ABB RAPID module: robotcode.MOD

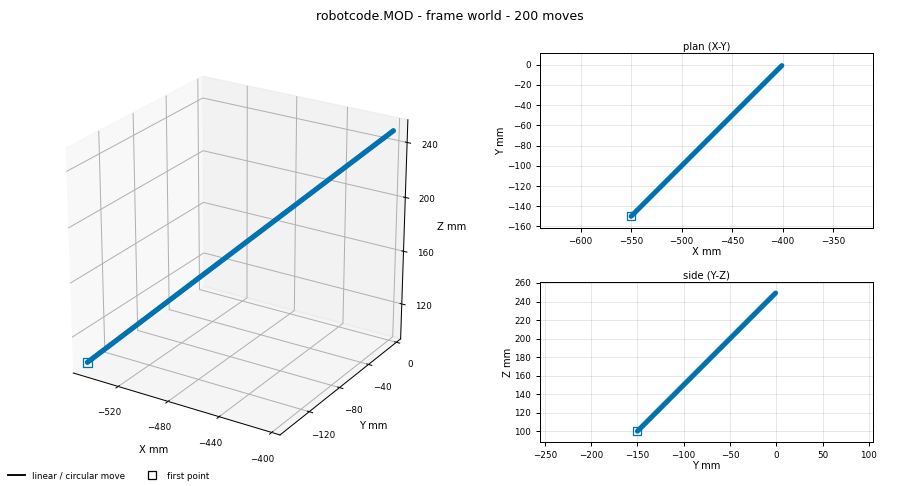
[picture p0: tool path of robotcode.MOD in frame world, 200 of 201 moves have a stored position in this frame; points joined in program order, loops and branches not executed]
MODULE MainModule
PERS tooldata Servo:=[TRUE,[[0,0,114.2],[1,0,0,0]],[0.215,[8.7,12.3,49.2],[1,0,0,0],0.00021,0.00024,0.00009]];
PERS tooldata tObject:=[TRUE,[[0,0,130],[0.707106781,-0.707106781,0,0]],[0.215,[8.7,12.3,49.2],[1,0,0,0],0.00021,0.00024,0.00009]];
PERS wobjdata handpos:= [FALSE,TRUE,"",[[-400,0,250],[1,0,0,0]],[[0,0,0],[1,0,0,0]]];
    PROC main()
        ConfL\Off;
        SingArea\Wrist;
        !Startpos
        MoveAbsJ [[0.441359,-16.418,10.8814,2.79121,60.2034,-14.3875],[168.362,9E+09,9E+09,9E+09,9E+09,9E+09]] \NoEOffs, v1000, fine, wi_tGripper;
        path;
    ENDPROC
    PROC path()

VAR robtarget t0 := [[-150.0, -150.0, -150.0], [0, -1, 0, 0], [0,0,-1,4], [-96,9E+09,9E+09,9E+09,9E+09,9E+09]];
VAR robtarget t1 := [[-149.25, -149.25, -149.25], [0, -1, 0, 0], [0,0,-1,4], [-96,9E+09,9E+09,9E+09,9E+09,9E+09]];
VAR robtarget t2 := [[-148.5, -148.5, -148.5], [0, -1, 0, 0], [0,0,-1,4], [-96,9E+09,9E+09,9E+09,9E+09,9E+09]];
VAR robtarget t3 := [[-147.75, -147.75, -147.75], [0, -1, 0, 0], [0,0,-1,4], [-96,9E+09,9E+09,9E+09,9E+09,9E+09]];
VAR robtarget t4 := [[-147.0, -147.0, -147.0], [0, -1, 0, 0], [0,0,-1,4], [-96,9E+09,9E+09,9E+09,9E+09,9E+09]];
VAR robtarget t5 := [[-146.25, -146.25, -146.25], [0, -1, 0, 0], [0,0,-1,4], [-96,9E+09,9E+09,9E+09,9E+09,9E+09]];
VAR robtarget t6 := [[-145.5, -145.5, -145.5], [0, -1, 0, 0], [0,0,-1,4], [-96,9E+09,9E+09,9E+09,9E+09,9E+09]];
VAR robtarget t7 := [[-144.75, -144.75, -144.75], [0, -1, 0, 0], [0,0,-1,4], [-96,9E+09,9E+09,9E+09,9E+09,9E+09]];
VAR robtarget t8 := [[-144.0, -144.0, -144.0], [0, -1, 0, 0], [0,0,-1,4], [-96,9E+09,9E+09,9E+09,9E+09,9E+09]];
VAR robtarget t9 := [[-143.25, -143.25, -143.25], [0, -1, 0, 0], [0,0,-1,4], [-96,9E+09,9E+09,9E+09,9E+09,9E+09]];
VAR robtarget t10 := [[-142.5, -142.5, -142.5], [0, -1, 0, 0], [0,0,-1,4], [-96,9E+09,9E+09,9E+09,9E+09,9E+09]];
VAR robtarget t11 := [[-141.75, -141.75, -141.75], [0, -1, 0, 0], [0,0,-1,4], [-96,9E+09,9E+09,9E+09,9E+09,9E+09]];
VAR robtarget t12 := [[-141.0, -141.0, -141.0], [0, -1, 0, 0], [0,0,-1,4], [-96,9E+09,9E+09,9E+09,9E+09,9E+09]];
VAR robtarget t13 := [[-140.25, -140.25, -140.25], [0, -1, 0, 0], [0,0,-1,4], [-96,9E+09,9E+09,9E+09,9E+09,9E+09]];
VAR robtarget t14 := [[-139.49999999999997, -139.49999999999997, -139.49999999999997], [0, -1, 0, 0], [0,0,-1,4], [-96,9E+09,9E+09,9E+09,9E+09,9E+09]];
VAR robtarget t15 := [[-138.74999999999997, -138.74999999999997, -138.74999999999997], [0, -1, 0, 0], [0,0,-1,4], [-96,9E+09,9E+09,9E+09,9E+09,9E+09]];
VAR robtarget t16 := [[-137.99999999999997, -137.99999999999997, -137.99999999999997], [0, -1, 0, 0], [0,0,-1,4], [-96,9E+09,9E+09,9E+09,9E+09,9E+09]];
VAR robtarget t17 := [[-137.24999999999997, -137.24999999999997, -137.24999999999997], [0, -1, 0, 0], [0,0,-1,4], [-96,9E+09,9E+09,9E+09,9E+09,9E+09]];
VAR robtarget t18 := [[-136.49999999999997, -136.49999999999997, -136.49999999999997], [0, -1, 0, 0], [0,0,-1,4], [-96,9E+09,9E+09,9E+09,9E+09,9E+09]];
VAR robtarget t19 := [[-135.74999999999997, -135.74999999999997, -135.74999999999997], [0, -1, 0, 0], [0,0,-1,4], [-96,9E+09,9E+09,9E+09,9E+09,9E+09]];
VAR robtarget t20 := [[-135.0, -135.0, -135.0], [0, -1, 0, 0], [0,0,-1,4], [-96,9E+09,9E+09,9E+09,9E+09,9E+09]];
VAR robtarget t21 := [[-134.24999999999997, -134.24999999999997, -134.24999999999997], [0, -1, 0, 0], [0,0,-1,4], [-96,9E+09,9E+09,9E+09,9E+09,9E+09]];
VAR robtarget t22 := [[-133.5, -133.5, -133.5], [0, -1, 0, 0], [0,0,-1,4], [-96,9E+09,9E+09,9E+09,9E+09,9E+09]];
VAR robtarget t23 := [[-132.74999999999997, -132.74999999999997, -132.74999999999997], [0, -1, 0, 0], [0,0,-1,4], [-96,9E+09,9E+09,9E+09,9E+09,9E+09]];
VAR robtarget t24 := [[-132.0, -132.0, -132.0], [0, -1, 0, 0], [0,0,-1,4], [-96,9E+09,9E+09,9E+09,9E+09,9E+09]];
VAR robtarget t25 := [[-131.25, -131.25, -131.25], [0, -1, 0, 0], [0,0,-1,4], [-96,9E+09,9E+09,9E+09,9E+09,9E+09]];
VAR robtarget t26 := [[-130.5, -130.5, -130.5], [0, -1, 0, 0], [0,0,-1,4], [-96,9E+09,9E+09,9E+09,9E+09,9E+09]];
VAR robtarget t27 := [[-129.75, -129.75, -129.75], [0, -1, 0, 0], [0,0,-1,4], [-96,9E+09,9E+09,9E+09,9E+09,9E+09]];
VAR robtarget t28 := [[-129.0, -129.0, -129.0], [0, -1, 0, 0], [0,0,-1,4], [-96,9E+09,9E+09,9E+09,9E+09,9E+09]];
VAR robtarget t29 := [[-128.25, -128.25, -128.25], [0, -1, 0, 0], [0,0,-1,4], [-96,9E+09,9E+09,9E+09,9E+09,9E+09]];
VAR robtarget t30 := [[-127.5, -127.5, -127.5], [0, -1, 0, 0], [0,0,-1,4], [-96,9E+09,9E+09,9E+09,9E+09,9E+09]];
VAR robtarget t31 := [[-126.75, -126.75, -126.75], [0, -1, 0, 0], [0,0,-1,4], [-96,9E+09,9E+09,9E+09,9E+09,9E+09]];
VAR robtarget t32 := [[-126.0, -126.0, -126.0], [0, -1, 0, 0], [0,0,-1,4], [-96,9E+09,9E+09,9E+09,9E+09,9E+09]];
VAR robtarget t33 := [[-125.25, -125.25, -125.25], [0, -1, 0, 0], [0,0,-1,4], [-96,9E+09,9E+09,9E+09,9E+09,9E+09]];
VAR robtarget t34 := [[-124.5, -124.5, -124.5], [0, -1, 0, 0], [0,0,-1,4], [-96,9E+09,9E+09,9E+09,9E+09,9E+09]];
VAR robtarget t35 := [[-123.75, -123.75, -123.75], [0, -1, 0, 0], [0,0,-1,4], [-96,9E+09,9E+09,9E+09,9E+09,9E+09]];
VAR robtarget t36 := [[-123.0, -123.0, -123.0], [0, -1, 0, 0], [0,0,-1,4], [-96,9E+09,9E+09,9E+09,9E+09,9E+09]];
VAR robtarget t37 := [[-122.25, -122.25, -122.25], [0, -1, 0, 0], [0,0,-1,4], [-96,9E+09,9E+09,9E+09,9E+09,9E+09]];
VAR robtarget t38 := [[-121.5, -121.5, -121.5], [0, -1, 0, 0], [0,0,-1,4], [-96,9E+09,9E+09,9E+09,9E+09,9E+09]];
VAR robtarget t39 := [[-120.75, -120.75, -120.75], [0, -1, 0, 0], [0,0,-1,4], [-96,9E+09,9E+09,9E+09,9E+09,9E+09]];
VAR robtarget t40 := [[-120.0, -120.0, -120.0], [0, -1, 0, 0], [0,0,-1,4], [-96,9E+09,9E+09,9E+09,9E+09,9E+09]];
VAR robtarget t41 := [[-119.25, -119.25, -119.25], [0, -1, 0, 0], [0,0,-1,4], [-96,9E+09,9E+09,9E+09,9E+09,9E+09]];
VAR robtarget t42 := [[-118.5, -118.5, -118.5], [0, -1, 0, 0], [0,0,-1,4], [-96,9E+09,9E+09,9E+09,9E+09,9E+09]];
VAR robtarget t43 := [[-117.75, -117.75, -117.75], [0, -1, 0, 0], [0,0,-1,4], [-96,9E+09,9E+09,9E+09,9E+09,9E+09]];
VAR robtarget t44 := [[-117.0, -117.0, -117.0], [0, -1, 0, 0], [0,0,-1,4], [-96,9E+09,9E+09,9E+09,9E+09,9E+09]];
VAR robtarget t45 := [[-116.24999999999999, -116.24999999999999, -116.24999999999999], [0, -1, 0, 0], [0,0,-1,4], [-96,9E+09,9E+09,9E+09,9E+09,9E+09]];
VAR robtarget t46 := [[-115.49999999999999, -115.49999999999999, -115.49999999999999], [0, -1, 0, 0], [0,0,-1,4], [-96,9E+09,9E+09,9E+09,9E+09,9E+09]];
VAR robtarget t47 := [[-114.74999999999999, -114.74999999999999, -114.74999999999999], [0, -1, 0, 0], [0,0,-1,4], [-96,9E+09,9E+09,9E+09,9E+09,9E+09]];
VAR robtarget t48 := [[-113.99999999999999, -113.99999999999999, -113.99999999999999], [0, -1, 0, 0], [0,0,-1,4], [-96,9E+09,9E+09,9E+09,9E+09,9E+09]];
VAR robtarget t49 := [[-113.24999999999999, -113.24999999999999, -113.24999999999999], [0, -1, 0, 0], [0,0,-1,4], [-96,9E+09,9E+09,9E+09,9E+09,9E+09]];
VAR robtarget t50 := [[-112.49999999999999, -112.49999999999999, -112.49999999999999], [0, -1, 0, 0], [0,0,-1,4], [-96,9E+09,9E+09,9E+09,9E+09,9E+09]];
VAR robtarget t51 := [[-111.74999999999999, -111.74999999999999, -111.74999999999999], [0, -1, 0, 0], [0,0,-1,4], [-96,9E+09,9E+09,9E+09,9E+09,9E+09]];
VAR robtarget t52 := [[-110.99999999999999, -110.99999999999999, -110.99999999999999], [0, -1, 0, 0], [0,0,-1,4], [-96,9E+09,9E+09,9E+09,9E+09,9E+09]];
VAR robtarget t53 := [[-110.24999999999999, -110.24999999999999, -110.24999999999999], [0, -1, 0, 0], [0,0,-1,4], [-96,9E+09,9E+09,9E+09,9E+09,9E+09]];
VAR robtarget t54 := [[-109.49999999999999, -109.49999999999999, -109.49999999999999], [0, -1, 0, 0], [0,0,-1,4], [-96,9E+09,9E+09,9E+09,9E+09,9E+09]];
VAR robtarget t55 := [[-108.74999999999999, -108.74999999999999, -108.74999999999999], [0, -1, 0, 0], [0,0,-1,4], [-96,9E+09,9E+09,9E+09,9E+09,9E+09]];
VAR robtarget t56 := [[-107.99999999999999, -107.99999999999999, -107.99999999999999], [0, -1, 0, 0], [0,0,-1,4], [-96,9E+09,9E+09,9E+09,9E+09,9E+09]];
VAR robtarget t57 := [[-107.24999999999999, -107.24999999999999, -107.24999999999999], [0, -1, 0, 0], [0,0,-1,4], [-96,9E+09,9E+09,9E+09,9E+09,9E+09]];
VAR robtarget t58 := [[-106.49999999999999, -106.49999999999999, -106.49999999999999], [0, -1, 0, 0], [0,0,-1,4], [-96,9E+09,9E+09,9E+09,9E+09,9E+09]];
VAR robtarget t59 := [[-105.75000000000001, -105.75000000000001, -105.75000000000001], [0, -1, 0, 0], [0,0,-1,4], [-96,9E+09,9E+09,9E+09,9E+09,9E+09]];
VAR robtarget t60 := [[-104.99999999999999, -104.99999999999999, -104.99999999999999], [0, -1, 0, 0], [0,0,-1,4], [-96,9E+09,9E+09,9E+09,9E+09,9E+09]];
VAR robtarget t61 := [[-104.25000000000001, -104.25000000000001, -104.25000000000001], [0, -1, 0, 0], [0,0,-1,4], [-96,9E+09,9E+09,9E+09,9E+09,9E+09]];
VAR robtarget t62 := [[-103.49999999999999, -103.49999999999999, -103.49999999999999], [0, -1, 0, 0], [0,0,-1,4], [-96,9E+09,9E+09,9E+09,9E+09,9E+09]];
VAR robtarget t63 := [[-102.75000000000001, -102.75000000000001, -102.75000000000001], [0, -1, 0, 0], [0,0,-1,4], [-96,9E+09,9E+09,9E+09,9E+09,9E+09]];
VAR robtarget t64 := [[-101.99999999999999, -101.99999999999999, -101.99999999999999], [0, -1, 0, 0], [0,0,-1,4], [-96,9E+09,9E+09,9E+09,9E+09,9E+09]];
VAR robtarget t65 := [[-101.25, -101.25, -101.25], [0, -1, 0, 0], [0,0,-1,4], [-96,9E+09,9E+09,9E+09,9E+09,9E+09]];
VAR robtarget t66 := [[-100.49999999999997, -100.49999999999997, -100.49999999999997], [0, -1, 0, 0], [0,0,-1,4], [-96,9E+09,9E+09,9E+09,9E+09,9E+09]];
VAR robtarget t67 := [[-99.75, -99.75, -99.75], [0, -1, 0, 0], [0,0,-1,4], [-96,9E+09,9E+09,9E+09,9E+09,9E+09]];
VAR robtarget t68 := [[-98.99999999999997, -98.99999999999997, -98.99999999999997], [0, -1, 0, 0], [0,0,-1,4], [-96,9E+09,9E+09,9E+09,9E+09,9E+09]];
VAR robtarget t69 := [[-98.25, -98.25, -98.25], [0, -1, 0, 0], [0,0,-1,4], [-96,9E+09,9E+09,9E+09,9E+09,9E+09]];
VAR robtarget t70 := [[-97.5, -97.5, -97.5], [0, -1, 0, 0], [0,0,-1,4], [-96,9E+09,9E+09,9E+09,9E+09,9E+09]];
VAR robtarget t71 := [[-96.75, -96.75, -96.75], [0, -1, 0, 0], [0,0,-1,4], [-96,9E+09,9E+09,9E+09,9E+09,9E+09]];
VAR robtarget t72 := [[-96.0, -96.0, -96.0], [0, -1, 0, 0], [0,0,-1,4], [-96,9E+09,9E+09,9E+09,9E+09,9E+09]];
VAR robtarget t73 := [[-95.25, -95.25, -95.25], [0, -1, 0, 0], [0,0,-1,4], [-96,9E+09,9E+09,9E+09,9E+09,9E+09]];
VAR robtarget t74 := [[-94.5, -94.5, -94.5], [0, -1, 0, 0], [0,0,-1,4], [-96,9E+09,9E+09,9E+09,9E+09,9E+09]];
VAR robtarget t75 := [[-93.75, -93.75, -93.75], [0, -1, 0, 0], [0,0,-1,4], [-96,9E+09,9E+09,9E+09,9E+09,9E+09]];
VAR robtarget t76 := [[-93.0, -93.0, -93.0], [0, -1, 0, 0], [0,0,-1,4], [-96,9E+09,9E+09,9E+09,9E+09,9E+09]];
VAR robtarget t77 := [[-92.25, -92.25, -92.25], [0, -1, 0, 0], [0,0,-1,4], [-96,9E+09,9E+09,9E+09,9E+09,9E+09]];
VAR robtarget t78 := [[-91.5, -91.5, -91.5], [0, -1, 0, 0], [0,0,-1,4], [-96,9E+09,9E+09,9E+09,9E+09,9E+09]];
VAR robtarget t79 := [[-90.75, -90.75, -90.75], [0, -1, 0, 0], [0,0,-1,4], [-96,9E+09,9E+09,9E+09,9E+09,9E+09]];
VAR robtarget t80 := [[-90.0, -90.0, -90.0], [0, -1, 0, 0], [0,0,-1,4], [-96,9E+09,9E+09,9E+09,9E+09,9E+09]];
VAR robtarget t81 := [[-89.25, -89.25, -89.25], [0, -1, 0, 0], [0,0,-1,4], [-96,9E+09,9E+09,9E+09,9E+09,9E+09]];
VAR robtarget t82 := [[-88.5, -88.5, -88.5], [0, -1, 0, 0], [0,0,-1,4], [-96,9E+09,9E+09,9E+09,9E+09,9E+09]];
VAR robtarget t83 := [[-87.75, -87.75, -87.75], [0, -1, 0, 0], [0,0,-1,4], [-96,9E+09,9E+09,9E+09,9E+09,9E+09]];
VAR robtarget t84 := [[-87.0, -87.0, -87.0], [0, -1, 0, 0], [0,0,-1,4], [-96,9E+09,9E+09,9E+09,9E+09,9E+09]];
VAR robtarget t85 := [[-86.25, -86.25, -86.25], [0, -1, 0, 0], [0,0,-1,4], [-96,9E+09,9E+09,9E+09,9E+09,9E+09]];
VAR robtarget t86 := [[-85.49999999999999, -85.49999999999999, -85.49999999999999], [0, -1, 0, 0], [0,0,-1,4], [-96,9E+09,9E+09,9E+09,9E+09,9E+09]];
VAR robtarget t87 := [[-84.74999999999999, -84.74999999999999, -84.74999999999999], [0, -1, 0, 0], [0,0,-1,4], [-96,9E+09,9E+09,9E+09,9E+09,9E+09]];
VAR robtarget t88 := [[-83.99999999999999, -83.99999999999999, -83.99999999999999], [0, -1, 0, 0], [0,0,-1,4], [-96,9E+09,9E+09,9E+09,9E+09,9E+09]];
VAR robtarget t89 := [[-83.24999999999999, -83.24999999999999, -83.24999999999999], [0, -1, 0, 0], [0,0,-1,4], [-96,9E+09,9E+09,9E+09,9E+09,9E+09]];
VAR robtarget t90 := [[-82.49999999999999, -82.49999999999999, -82.49999999999999], [0, -1, 0, 0], [0,0,-1,4], [-96,9E+09,9E+09,9E+09,9E+09,9E+09]];
VAR robtarget t91 := [[-81.74999999999999, -81.74999999999999, -81.74999999999999], [0, -1, 0, 0], [0,0,-1,4], [-96,9E+09,9E+09,9E+09,9E+09,9E+09]];
VAR robtarget t92 := [[-80.99999999999999, -80.99999999999999, -80.99999999999999], [0, -1, 0, 0], [0,0,-1,4], [-96,9E+09,9E+09,9E+09,9E+09,9E+09]];
VAR robtarget t93 := [[-80.24999999999999, -80.24999999999999, -80.24999999999999], [0, -1, 0, 0], [0,0,-1,4], [-96,9E+09,9E+09,9E+09,9E+09,9E+09]];
VAR robtarget t94 := [[-79.49999999999999, -79.49999999999999, -79.49999999999999], [0, -1, 0, 0], [0,0,-1,4], [-96,9E+09,9E+09,9E+09,9E+09,9E+09]];
VAR robtarget t95 := [[-78.74999999999999, -78.74999999999999, -78.74999999999999], [0, -1, 0, 0], [0,0,-1,4], [-96,9E+09,9E+09,9E+09,9E+09,9E+09]];
VAR robtarget t96 := [[-77.99999999999999, -77.99999999999999, -77.99999999999999], [0, -1, 0, 0], [0,0,-1,4], [-96,9E+09,9E+09,9E+09,9E+09,9E+09]];
VAR robtarget t97 := [[-77.24999999999999, -77.24999999999999, -77.24999999999999], [0, -1, 0, 0], [0,0,-1,4], [-96,9E+09,9E+09,9E+09,9E+09,9E+09]];
VAR robtarget t98 := [[-76.50000000000001, -76.50000000000001, -76.50000000000001], [0, -1, 0, 0], [0,0,-1,4], [-96,9E+09,9E+09,9E+09,9E+09,9E+09]];
VAR robtarget t99 := [[-75.74999999999999, -75.74999999999999, -75.74999999999999], [0, -1, 0, 0], [0,0,-1,4], [-96,9E+09,9E+09,9E+09,9E+09,9E+09]];
VAR robtarget t100 := [[-75.00000000000001, -75.00000000000001, -75.00000000000001], [0, -1, 0, 0], [0,0,-1,4], [-96,9E+09,9E+09,9E+09,9E+09,9E+09]];
VAR robtarget t101 := [[-74.24999999999999, -74.24999999999999, -74.24999999999999], [0, -1, 0, 0], [0,0,-1,4], [-96,9E+09,9E+09,9E+09,9E+09,9E+09]];
VAR robtarget t102 := [[-73.50000000000001, -73.50000000000001, -73.50000000000001], [0, -1, 0, 0], [0,0,-1,4], [-96,9E+09,9E+09,9E+09,9E+09,9E+09]];
VAR robtarget t103 := [[-72.74999999999999, -72.74999999999999, -72.74999999999999], [0, -1, 0, 0], [0,0,-1,4], [-96,9E+09,9E+09,9E+09,9E+09,9E+09]];
VAR robtarget t104 := [[-72.00000000000001, -72.00000000000001, -72.00000000000001], [0, -1, 0, 0], [0,0,-1,4], [-96,9E+09,9E+09,9E+09,9E+09,9E+09]];
VAR robtarget t105 := [[-71.24999999999999, -71.24999999999999, -71.24999999999999], [0, -1, 0, 0], [0,0,-1,4], [-96,9E+09,9E+09,9E+09,9E+09,9E+09]];
VAR robtarget t106 := [[-70.5, -70.5, -70.5], [0, -1, 0, 0], [0,0,-1,4], [-96,9E+09,9E+09,9E+09,9E+09,9E+09]];
VAR robtarget t107 := [[-69.74999999999997, -69.74999999999997, -69.74999999999997], [0, -1, 0, 0], [0,0,-1,4], [-96,9E+09,9E+09,9E+09,9E+09,9E+09]];
VAR robtarget t108 := [[-69.0, -69.0, -69.0], [0, -1, 0, 0], [0,0,-1,4], [-96,9E+09,9E+09,9E+09,9E+09,9E+09]];
VAR robtarget t109 := [[-68.24999999999997, -68.24999999999997, -68.24999999999997], [0, -1, 0, 0], [0,0,-1,4], [-96,9E+09,9E+09,9E+09,9E+09,9E+09]];
VAR robtarget t110 := [[-67.5, -67.5, -67.5], [0, -1, 0, 0], [0,0,-1,4], [-96,9E+09,9E+09,9E+09,9E+09,9E+09]];
VAR robtarget t111 := [[-66.74999999999997, -66.74999999999997, -66.74999999999997], [0, -1, 0, 0], [0,0,-1,4], [-96,9E+09,9E+09,9E+09,9E+09,9E+09]];
VAR robtarget t112 := [[-66.0, -66.0, -66.0], [0, -1, 0, 0], [0,0,-1,4], [-96,9E+09,9E+09,9E+09,9E+09,9E+09]];
VAR robtarget t113 := [[-65.24999999999997, -65.24999999999997, -65.24999999999997], [0, -1, 0, 0], [0,0,-1,4], [-96,9E+09,9E+09,9E+09,9E+09,9E+09]];
VAR robtarget t114 := [[-64.5, -64.5, -64.5], [0, -1, 0, 0], [0,0,-1,4], [-96,9E+09,9E+09,9E+09,9E+09,9E+09]];
VAR robtarget t115 := [[-63.74999999999997, -63.74999999999997, -63.74999999999997], [0, -1, 0, 0], [0,0,-1,4], [-96,9E+09,9E+09,9E+09,9E+09,9E+09]];
VAR robtarget t116 := [[-63.0, -63.0, -63.0], [0, -1, 0, 0], [0,0,-1,4], [-96,9E+09,9E+09,9E+09,9E+09,9E+09]];
VAR robtarget t117 := [[-62.24999999999997, -62.24999999999997, -62.24999999999997], [0, -1, 0, 0], [0,0,-1,4], [-96,9E+09,9E+09,9E+09,9E+09,9E+09]];
VAR robtarget t118 := [[-61.5, -61.5, -61.5], [0, -1, 0, 0], [0,0,-1,4], [-96,9E+09,9E+09,9E+09,9E+09,9E+09]];
VAR robtarget t119 := [[-60.75, -60.75, -60.75], [0, -1, 0, 0], [0,0,-1,4], [-96,9E+09,9E+09,9E+09,9E+09,9E+09]];
VAR robtarget t120 := [[-60.0, -60.0, -60.0], [0, -1, 0, 0], [0,0,-1,4], [-96,9E+09,9E+09,9E+09,9E+09,9E+09]];
VAR robtarget t121 := [[-59.25, -59.25, -59.25], [0, -1, 0, 0], [0,0,-1,4], [-96,9E+09,9E+09,9E+09,9E+09,9E+09]];
VAR robtarget t122 := [[-58.5, -58.5, -58.5], [0, -1, 0, 0], [0,0,-1,4], [-96,9E+09,9E+09,9E+09,9E+09,9E+09]];
VAR robtarget t123 := [[-57.74999999999999, -57.74999999999999, -57.74999999999999], [0, -1, 0, 0], [0,0,-1,4], [-96,9E+09,9E+09,9E+09,9E+09,9E+09]];
VAR robtarget t124 := [[-56.99999999999999, -56.99999999999999, -56.99999999999999], [0, -1, 0, 0], [0,0,-1,4], [-96,9E+09,9E+09,9E+09,9E+09,9E+09]];
VAR robtarget t125 := [[-56.24999999999999, -56.24999999999999, -56.24999999999999], [0, -1, 0, 0], [0,0,-1,4], [-96,9E+09,9E+09,9E+09,9E+09,9E+09]];
VAR robtarget t126 := [[-55.49999999999999, -55.49999999999999, -55.49999999999999], [0, -1, 0, 0], [0,0,-1,4], [-96,9E+09,9E+09,9E+09,9E+09,9E+09]];
VAR robtarget t127 := [[-54.74999999999999, -54.74999999999999, -54.74999999999999], [0, -1, 0, 0], [0,0,-1,4], [-96,9E+09,9E+09,9E+09,9E+09,9E+09]];
VAR robtarget t128 := [[-53.99999999999999, -53.99999999999999, -53.99999999999999], [0, -1, 0, 0], [0,0,-1,4], [-96,9E+09,9E+09,9E+09,9E+09,9E+09]];
VAR robtarget t129 := [[-53.24999999999999, -53.24999999999999, -53.24999999999999], [0, -1, 0, 0], [0,0,-1,4], [-96,9E+09,9E+09,9E+09,9E+09,9E+09]];
VAR robtarget t130 := [[-52.49999999999999, -52.49999999999999, -52.49999999999999], [0, -1, 0, 0], [0,0,-1,4], [-96,9E+09,9E+09,9E+09,9E+09,9E+09]];
VAR robtarget t131 := [[-51.74999999999999, -51.74999999999999, -51.74999999999999], [0, -1, 0, 0], [0,0,-1,4], [-96,9E+09,9E+09,9E+09,9E+09,9E+09]];
VAR robtarget t132 := [[-50.99999999999999, -50.99999999999999, -50.99999999999999], [0, -1, 0, 0], [0,0,-1,4], [-96,9E+09,9E+09,9E+09,9E+09,9E+09]];
VAR robtarget t133 := [[-50.249999999999986, -50.249999999999986, -50.249999999999986], [0, -1, 0, 0], [0,0,-1,4], [-96,9E+09,9E+09,9E+09,9E+09,9E+09]];
VAR robtarget t134 := [[-49.499999999999986, -49.499999999999986, -49.499999999999986], [0, -1, 0, 0], [0,0,-1,4], [-96,9E+09,9E+09,9E+09,9E+09,9E+09]];
VAR robtarget t135 := [[-48.750000000000014, -48.750000000000014, -48.750000000000014], [0, -1, 0, 0], [0,0,-1,4], [-96,9E+09,9E+09,9E+09,9E+09,9E+09]];
VAR robtarget t136 := [[-47.999999999999986, -47.999999999999986, -47.999999999999986], [0, -1, 0, 0], [0,0,-1,4], [-96,9E+09,9E+09,9E+09,9E+09,9E+09]];
VAR robtarget t137 := [[-47.24999999999996, -47.24999999999996, -47.24999999999996], [0, -1, 0, 0], [0,0,-1,4], [-96,9E+09,9E+09,9E+09,9E+09,9E+09]];
VAR robtarget t138 := [[-46.499999999999986, -46.499999999999986, -46.499999999999986], [0, -1, 0, 0], [0,0,-1,4], [-96,9E+09,9E+09,9E+09,9E+09,9E+09]];
VAR robtarget t139 := [[-45.750000000000014, -45.750000000000014, -45.750000000000014], [0, -1, 0, 0], [0,0,-1,4], [-96,9E+09,9E+09,9E+09,9E+09,9E+09]];
VAR robtarget t140 := [[-44.999999999999986, -44.999999999999986, -44.999999999999986], [0, -1, 0, 0], [0,0,-1,4], [-96,9E+09,9E+09,9E+09,9E+09,9E+09]];
VAR robtarget t141 := [[-44.250000000000014, -44.250000000000014, -44.250000000000014], [0, -1, 0, 0], [0,0,-1,4], [-96,9E+09,9E+09,9E+09,9E+09,9E+09]];
VAR robtarget t142 := [[-43.499999999999986, -43.499999999999986, -43.499999999999986], [0, -1, 0, 0], [0,0,-1,4], [-96,9E+09,9E+09,9E+09,9E+09,9E+09]];
VAR robtarget t143 := [[-42.75000000000001, -42.75000000000001, -42.75000000000001], [0, -1, 0, 0], [0,0,-1,4], [-96,9E+09,9E+09,9E+09,9E+09,9E+09]];
VAR robtarget t144 := [[-41.99999999999998, -41.99999999999998, -41.99999999999998], [0, -1, 0, 0], [0,0,-1,4], [-96,9E+09,9E+09,9E+09,9E+09,9E+09]];
VAR robtarget t145 := [[-41.25000000000001, -41.25000000000001, -41.25000000000001], [0, -1, 0, 0], [0,0,-1,4], [-96,9E+09,9E+09,9E+09,9E+09,9E+09]];
VAR robtarget t146 := [[-40.49999999999998, -40.49999999999998, -40.49999999999998], [0, -1, 0, 0], [0,0,-1,4], [-96,9E+09,9E+09,9E+09,9E+09,9E+09]];
VAR robtarget t147 := [[-39.75000000000001, -39.75000000000001, -39.75000000000001], [0, -1, 0, 0], [0,0,-1,4], [-96,9E+09,9E+09,9E+09,9E+09,9E+09]];
VAR robtarget t148 := [[-38.99999999999998, -38.99999999999998, -38.99999999999998], [0, -1, 0, 0], [0,0,-1,4], [-96,9E+09,9E+09,9E+09,9E+09,9E+09]];
VAR robtarget t149 := [[-38.25000000000001, -38.25000000000001, -38.25000000000001], [0, -1, 0, 0], [0,0,-1,4], [-96,9E+09,9E+09,9E+09,9E+09,9E+09]];
VAR robtarget t150 := [[-37.49999999999998, -37.49999999999998, -37.49999999999998], [0, -1, 0, 0], [0,0,-1,4], [-96,9E+09,9E+09,9E+09,9E+09,9E+09]];
VAR robtarget t151 := [[-36.75000000000001, -36.75000000000001, -36.75000000000001], [0, -1, 0, 0], [0,0,-1,4], [-96,9E+09,9E+09,9E+09,9E+09,9E+09]];
VAR robtarget t152 := [[-35.99999999999998, -35.99999999999998, -35.99999999999998], [0, -1, 0, 0], [0,0,-1,4], [-96,9E+09,9E+09,9E+09,9E+09,9E+09]];
VAR robtarget t153 := [[-35.25, -35.25, -35.25], [0, -1, 0, 0], [0,0,-1,4], [-96,9E+09,9E+09,9E+09,9E+09,9E+09]];
VAR robtarget t154 := [[-34.49999999999997, -34.49999999999997, -34.49999999999997], [0, -1, 0, 0], [0,0,-1,4], [-96,9E+09,9E+09,9E+09,9E+09,9E+09]];
VAR robtarget t155 := [[-33.75, -33.75, -33.75], [0, -1, 0, 0], [0,0,-1,4], [-96,9E+09,9E+09,9E+09,9E+09,9E+09]];
VAR robtarget t156 := [[-32.99999999999997, -32.99999999999997, -32.99999999999997], [0, -1, 0, 0], [0,0,-1,4], [-96,9E+09,9E+09,9E+09,9E+09,9E+09]];
VAR robtarget t157 := [[-32.25, -32.25, -32.25], [0, -1, 0, 0], [0,0,-1,4], [-96,9E+09,9E+09,9E+09,9E+09,9E+09]];
VAR robtarget t158 := [[-31.49999999999997, -31.49999999999997, -31.49999999999997], [0, -1, 0, 0], [0,0,-1,4], [-96,9E+09,9E+09,9E+09,9E+09,9E+09]];
VAR robtarget t159 := [[-30.75, -30.75, -30.75], [0, -1, 0, 0], [0,0,-1,4], [-96,9E+09,9E+09,9E+09,9E+09,9E+09]];
VAR robtarget t160 := [[-29.99999999999997, -29.99999999999997, -29.99999999999997], [0, -1, 0, 0], [0,0,-1,4], [-96,9E+09,9E+09,9E+09,9E+09,9E+09]];
VAR robtarget t161 := [[-29.25, -29.25, -29.25], [0, -1, 0, 0], [0,0,-1,4], [-96,9E+09,9E+09,9E+09,9E+09,9E+09]];
VAR robtarget t162 := [[-28.500000000000025, -28.500000000000025, -28.500000000000025], [0, -1, 0, 0], [0,0,-1,4], [-96,9E+09,9E+09,9E+09,9E+09,9E+09]];
VAR robtarget t163 := [[-27.749999999999996, -27.749999999999996, -27.749999999999996], [0, -1, 0, 0], [0,0,-1,4], [-96,9E+09,9E+09,9E+09,9E+09,9E+09]];
VAR robtarget t164 := [[-26.999999999999968, -26.999999999999968, -26.999999999999968], [0, -1, 0, 0], [0,0,-1,4], [-96,9E+09,9E+09,9E+09,9E+09,9E+09]];
VAR robtarget t165 := [[-26.249999999999996, -26.249999999999996, -26.249999999999996], [0, -1, 0, 0], [0,0,-1,4], [-96,9E+09,9E+09,9E+09,9E+09,9E+09]];
VAR robtarget t166 := [[-25.50000000000002, -25.50000000000002, -25.50000000000002], [0, -1, 0, 0], [0,0,-1,4], [-96,9E+09,9E+09,9E+09,9E+09,9E+09]];
VAR robtarget t167 := [[-24.749999999999993, -24.749999999999993, -24.749999999999993], [0, -1, 0, 0], [0,0,-1,4], [-96,9E+09,9E+09,9E+09,9E+09,9E+09]];
VAR robtarget t168 := [[-23.999999999999964, -23.999999999999964, -23.999999999999964], [0, -1, 0, 0], [0,0,-1,4], [-96,9E+09,9E+09,9E+09,9E+09,9E+09]];
VAR robtarget t169 := [[-23.249999999999993, -23.249999999999993, -23.249999999999993], [0, -1, 0, 0], [0,0,-1,4], [-96,9E+09,9E+09,9E+09,9E+09,9E+09]];
VAR robtarget t170 := [[-22.50000000000002, -22.50000000000002, -22.50000000000002], [0, -1, 0, 0], [0,0,-1,4], [-96,9E+09,9E+09,9E+09,9E+09,9E+09]];
VAR robtarget t171 := [[-21.749999999999993, -21.749999999999993, -21.749999999999993], [0, -1, 0, 0], [0,0,-1,4], [-96,9E+09,9E+09,9E+09,9E+09,9E+09]];
VAR robtarget t172 := [[-20.999999999999964, -20.999999999999964, -20.999999999999964], [0, -1, 0, 0], [0,0,-1,4], [-96,9E+09,9E+09,9E+09,9E+09,9E+09]];
VAR robtarget t173 := [[-20.24999999999999, -20.24999999999999, -20.24999999999999], [0, -1, 0, 0], [0,0,-1,4], [-96,9E+09,9E+09,9E+09,9E+09,9E+09]];
VAR robtarget t174 := [[-19.500000000000018, -19.500000000000018, -19.500000000000018], [0, -1, 0, 0], [0,0,-1,4], [-96,9E+09,9E+09,9E+09,9E+09,9E+09]];
VAR robtarget t175 := [[-18.74999999999999, -18.74999999999999, -18.74999999999999], [0, -1, 0, 0], [0,0,-1,4], [-96,9E+09,9E+09,9E+09,9E+09,9E+09]];
VAR robtarget t176 := [[-17.99999999999996, -17.99999999999996, -17.99999999999996], [0, -1, 0, 0], [0,0,-1,4], [-96,9E+09,9E+09,9E+09,9E+09,9E+09]];
VAR robtarget t177 := [[-17.249999999999986, -17.249999999999986, -17.249999999999986], [0, -1, 0, 0], [0,0,-1,4], [-96,9E+09,9E+09,9E+09,9E+09,9E+09]];
VAR robtarget t178 := [[-16.500000000000014, -16.500000000000014, -16.500000000000014], [0, -1, 0, 0], [0,0,-1,4], [-96,9E+09,9E+09,9E+09,9E+09,9E+09]];
VAR robtarget t179 := [[-15.749999999999986, -15.749999999999986, -15.749999999999986], [0, -1, 0, 0], [0,0,-1,4], [-96,9E+09,9E+09,9E+09,9E+09,9E+09]];
VAR robtarget t180 := [[-14.999999999999957, -14.999999999999957, -14.999999999999957], [0, -1, 0, 0], [0,0,-1,4], [-96,9E+09,9E+09,9E+09,9E+09,9E+09]];
VAR robtarget t181 := [[-14.249999999999986, -14.249999999999986, -14.249999999999986], [0, -1, 0, 0], [0,0,-1,4], [-96,9E+09,9E+09,9E+09,9E+09,9E+09]];
VAR robtarget t182 := [[-13.500000000000012, -13.500000000000012, -13.500000000000012], [0, -1, 0, 0], [0,0,-1,4], [-96,9E+09,9E+09,9E+09,9E+09,9E+09]];
VAR robtarget t183 := [[-12.749999999999984, -12.749999999999984, -12.749999999999984], [0, -1, 0, 0], [0,0,-1,4], [-96,9E+09,9E+09,9E+09,9E+09,9E+09]];
VAR robtarget t184 := [[-11.999999999999956, -11.999999999999956, -11.999999999999956], [0, -1, 0, 0], [0,0,-1,4], [-96,9E+09,9E+09,9E+09,9E+09,9E+09]];
VAR robtarget t185 := [[-11.249999999999982, -11.249999999999982, -11.249999999999982], [0, -1, 0, 0], [0,0,-1,4], [-96,9E+09,9E+09,9E+09,9E+09,9E+09]];
VAR robtarget t186 := [[-10.500000000000009, -10.500000000000009, -10.500000000000009], [0, -1, 0, 0], [0,0,-1,4], [-96,9E+09,9E+09,9E+09,9E+09,9E+09]];
VAR robtarget t187 := [[-9.74999999999998, -9.74999999999998, -9.74999999999998], [0, -1, 0, 0], [0,0,-1,4], [-96,9E+09,9E+09,9E+09,9E+09,9E+09]];
VAR robtarget t188 := [[-8.999999999999952, -8.999999999999952, -8.999999999999952], [0, -1, 0, 0], [0,0,-1,4], [-96,9E+09,9E+09,9E+09,9E+09,9E+09]];
VAR robtarget t189 := [[-8.249999999999979, -8.249999999999979, -8.249999999999979], [0, -1, 0, 0], [0,0,-1,4], [-96,9E+09,9E+09,9E+09,9E+09,9E+09]];
VAR robtarget t190 := [[-7.500000000000007, -7.500000000000007, -7.500000000000007], [0, -1, 0, 0], [0,0,-1,4], [-96,9E+09,9E+09,9E+09,9E+09,9E+09]];
VAR robtarget t191 := [[-6.749999999999979, -6.749999999999979, -6.749999999999979], [0, -1, 0, 0], [0,0,-1,4], [-96,9E+09,9E+09,9E+09,9E+09,9E+09]];
VAR robtarget t192 := [[-5.99999999999995, -5.99999999999995, -5.99999999999995], [0, -1, 0, 0], [0,0,-1,4], [-96,9E+09,9E+09,9E+09,9E+09,9E+09]];
VAR robtarget t193 := [[-5.250000000000032, -5.250000000000032, -5.250000000000032], [0, -1, 0, 0], [0,0,-1,4], [-96,9E+09,9E+09,9E+09,9E+09,9E+09]];
VAR robtarget t194 := [[-4.5000000000000036, -4.5000000000000036, -4.5000000000000036], [0, -1, 0, 0], [0,0,-1,4], [-96,9E+09,9E+09,9E+09,9E+09,9E+09]];
VAR robtarget t195 := [[-3.7499999999999756, -3.7499999999999756, -3.7499999999999756], [0, -1, 0, 0], [0,0,-1,4], [-96,9E+09,9E+09,9E+09,9E+09,9E+09]];
VAR robtarget t196 := [[-3.0000000000000027, -3.0000000000000027, -3.0000000000000027], [0, -1, 0, 0], [0,0,-1,4], [-96,9E+09,9E+09,9E+09,9E+09,9E+09]];
VAR robtarget t197 := [[-2.2500000000000298, -2.2500000000000298, -2.2500000000000298], [0, -1, 0, 0], [0,0,-1,4], [-96,9E+09,9E+09,9E+09,9E+09,9E+09]];
VAR robtarget t198 := [[-1.5000000000000013, -1.5000000000000013, -1.5000000000000013], [0, -1, 0, 0], [0,0,-1,4], [-96,9E+09,9E+09,9E+09,9E+09,9E+09]];
VAR robtarget t199 := [[-0.7499999999999729, -0.7499999999999729, -0.7499999999999729], [0, -1, 0, 0], [0,0,-1,4], [-96,9E+09,9E+09,9E+09,9E+09,9E+09]];MoveL t0, v100\V:=100.000, z1, wi_tGripper, \WObj:=handpos;
MoveL t1, v100\V:=100.000, z1, wi_tGripper, \WObj:=handpos;
MoveL t2, v100\V:=100.000, z1, wi_tGripper, \WObj:=handpos;
MoveL t3, v100\V:=100.000, z1, wi_tGripper, \WObj:=handpos;
MoveL t4, v100\V:=100.000, z1, wi_tGripper, \WObj:=handpos;
MoveL t5, v100\V:=100.000, z1, wi_tGripper, \WObj:=handpos;
MoveL t6, v100\V:=100.000, z1, wi_tGripper, \WObj:=handpos;
MoveL t7, v100\V:=100.000, z1, wi_tGripper, \WObj:=handpos;
MoveL t8, v100\V:=100.000, z1, wi_tGripper, \WObj:=handpos;
MoveL t9, v100\V:=100.000, z1, wi_tGripper, \WObj:=handpos;
MoveL t10, v100\V:=100.000, z1, wi_tGripper, \WObj:=handpos;
MoveL t11, v100\V:=100.000, z1, wi_tGripper, \WObj:=handpos;
MoveL t12, v100\V:=100.000, z1, wi_tGripper, \WObj:=handpos;
MoveL t13, v100\V:=100.000, z1, wi_tGripper, \WObj:=handpos;
MoveL t14, v100\V:=100.000, z1, wi_tGripper, \WObj:=handpos;
MoveL t15, v100\V:=100.000, z1, wi_tGripper, \WObj:=handpos;
MoveL t16, v100\V:=100.000, z1, wi_tGripper, \WObj:=handpos;
MoveL t17, v100\V:=100.000, z1, wi_tGripper, \WObj:=handpos;
MoveL t18, v100\V:=100.000, z1, wi_tGripper, \WObj:=handpos;
MoveL t19, v100\V:=100.000, z1, wi_tGripper, \WObj:=handpos;
MoveL t20, v100\V:=100.000, z1, wi_tGripper, \WObj:=handpos;
MoveL t21, v100\V:=100.000, z1, wi_tGripper, \WObj:=handpos;
MoveL t22, v100\V:=100.000, z1, wi_tGripper, \WObj:=handpos;
MoveL t23, v100\V:=100.000, z1, wi_tGripper, \WObj:=handpos;
MoveL t24, v100\V:=100.000, z1, wi_tGripper, \WObj:=handpos;
MoveL t25, v100\V:=100.000, z1, wi_tGripper, \WObj:=handpos;
MoveL t26, v100\V:=100.000, z1, wi_tGripper, \WObj:=handpos;
MoveL t27, v100\V:=100.000, z1, wi_tGripper, \WObj:=handpos;
MoveL t28, v100\V:=100.000, z1, wi_tGripper, \WObj:=handpos;
MoveL t29, v100\V:=100.000, z1, wi_tGripper, \WObj:=handpos;
MoveL t30, v100\V:=100.000, z1, wi_tGripper, \WObj:=handpos;
MoveL t31, v100\V:=100.000, z1, wi_tGripper, \WObj:=handpos;
MoveL t32, v100\V:=100.000, z1, wi_tGripper, \WObj:=handpos;
MoveL t33, v100\V:=100.000, z1, wi_tGripper, \WObj:=handpos;
MoveL t34, v100\V:=100.000, z1, wi_tGripper, \WObj:=handpos;
MoveL t35, v100\V:=100.000, z1, wi_tGripper, \WObj:=handpos;
MoveL t36, v100\V:=100.000, z1, wi_tGripper, \WObj:=handpos;
MoveL t37, v100\V:=100.000, z1, wi_tGripper, \WObj:=handpos;
MoveL t38, v100\V:=100.000, z1, wi_tGripper, \WObj:=handpos;
MoveL t39, v100\V:=100.000, z1, wi_tGripper, \WObj:=handpos;
MoveL t40, v100\V:=100.000, z1, wi_tGripper, \WObj:=handpos;
MoveL t41, v100\V:=100.000, z1, wi_tGripper, \WObj:=handpos;
MoveL t42, v100\V:=100.000, z1, wi_tGripper, \WObj:=handpos;
MoveL t43, v100\V:=100.000, z1, wi_tGripper, \WObj:=handpos;
MoveL t44, v100\V:=100.000, z1, wi_tGripper, \WObj:=handpos;
MoveL t45, v100\V:=100.000, z1, wi_tGripper, \WObj:=handpos;
MoveL t46, v100\V:=100.000, z1, wi_tGripper, \WObj:=handpos;
MoveL t47, v100\V:=100.000, z1, wi_tGripper, \WObj:=handpos;
MoveL t48, v100\V:=100.000, z1, wi_tGripper, \WObj:=handpos;
MoveL t49, v100\V:=100.000, z1, wi_tGripper, \WObj:=handpos;
MoveL t50, v100\V:=100.000, z1, wi_tGripper, \WObj:=handpos;
MoveL t51, v100\V:=100.000, z1, wi_tGripper, \WObj:=handpos;
MoveL t52, v100\V:=100.000, z1, wi_tGripper, \WObj:=handpos;
MoveL t53, v100\V:=100.000, z1, wi_tGripper, \WObj:=handpos;
MoveL t54, v100\V:=100.000, z1, wi_tGripper, \WObj:=handpos;
MoveL t55, v100\V:=100.000, z1, wi_tGripper, \WObj:=handpos;
MoveL t56, v100\V:=100.000, z1, wi_tGripper, \WObj:=handpos;
MoveL t57, v100\V:=100.000, z1, wi_tGripper, \WObj:=handpos;
MoveL t58, v100\V:=100.000, z1, wi_tGripper, \WObj:=handpos;
MoveL t59, v100\V:=100.000, z1, wi_tGripper, \WObj:=handpos;
MoveL t60, v100\V:=100.000, z1, wi_tGripper, \WObj:=handpos;
MoveL t61, v100\V:=100.000, z1, wi_tGripper, \WObj:=handpos;
MoveL t62, v100\V:=100.000, z1, wi_tGripper, \WObj:=handpos;
MoveL t63, v100\V:=100.000, z1, wi_tGripper, \WObj:=handpos;
MoveL t64, v100\V:=100.000, z1, wi_tGripper, \WObj:=handpos;
MoveL t65, v100\V:=100.000, z1, wi_tGripper, \WObj:=handpos;
MoveL t66, v100\V:=100.000, z1, wi_tGripper, \WObj:=handpos;
MoveL t67, v100\V:=100.000, z1, wi_tGripper, \WObj:=handpos;
MoveL t68, v100\V:=100.000, z1, wi_tGripper, \WObj:=handpos;
MoveL t69, v100\V:=100.000, z1, wi_tGripper, \WObj:=handpos;
MoveL t70, v100\V:=100.000, z1, wi_tGripper, \WObj:=handpos;
MoveL t71, v100\V:=100.000, z1, wi_tGripper, \WObj:=handpos;
MoveL t72, v100\V:=100.000, z1, wi_tGripper, \WObj:=handpos;
MoveL t73, v100\V:=100.000, z1, wi_tGripper, \WObj:=handpos;
MoveL t74, v100\V:=100.000, z1, wi_tGripper, \WObj:=handpos;
MoveL t75, v100\V:=100.000, z1, wi_tGripper, \WObj:=handpos;
MoveL t76, v100\V:=100.000, z1, wi_tGripper, \WObj:=handpos;
MoveL t77, v100\V:=100.000, z1, wi_tGripper, \WObj:=handpos;
MoveL t78, v100\V:=100.000, z1, wi_tGripper, \WObj:=handpos;
MoveL t79, v100\V:=100.000, z1, wi_tGripper, \WObj:=handpos;
MoveL t80, v100\V:=100.000, z1, wi_tGripper, \WObj:=handpos;
MoveL t81, v100\V:=100.000, z1, wi_tGripper, \WObj:=handpos;
MoveL t82, v100\V:=100.000, z1, wi_tGripper, \WObj:=handpos;
MoveL t83, v100\V:=100.000, z1, wi_tGripper, \WObj:=handpos;
MoveL t84, v100\V:=100.000, z1, wi_tGripper, \WObj:=handpos;
MoveL t85, v100\V:=100.000, z1, wi_tGripper, \WObj:=handpos;
MoveL t86, v100\V:=100.000, z1, wi_tGripper, \WObj:=handpos;
MoveL t87, v100\V:=100.000, z1, wi_tGripper, \WObj:=handpos;
MoveL t88, v100\V:=100.000, z1, wi_tGripper, \WObj:=handpos;
MoveL t89, v100\V:=100.000, z1, wi_tGripper, \WObj:=handpos;
MoveL t90, v100\V:=100.000, z1, wi_tGripper, \WObj:=handpos;
MoveL t91, v100\V:=100.000, z1, wi_tGripper, \WObj:=handpos;
MoveL t92, v100\V:=100.000, z1, wi_tGripper, \WObj:=handpos;
MoveL t93, v100\V:=100.000, z1, wi_tGripper, \WObj:=handpos;
MoveL t94, v100\V:=100.000, z1, wi_tGripper, \WObj:=handpos;
MoveL t95, v100\V:=100.000, z1, wi_tGripper, \WObj:=handpos;
MoveL t96, v100\V:=100.000, z1, wi_tGripper, \WObj:=handpos;
MoveL t97, v100\V:=100.000, z1, wi_tGripper, \WObj:=handpos;
MoveL t98, v100\V:=100.000, z1, wi_tGripper, \WObj:=handpos;
MoveL t99, v100\V:=100.000, z1, wi_tGripper, \WObj:=handpos;
MoveL t100, v100\V:=100.000, z1, wi_tGripper, \WObj:=handpos;
MoveL t101, v100\V:=100.000, z1, wi_tGripper, \WObj:=handpos;
MoveL t102, v100\V:=100.000, z1, wi_tGripper, \WObj:=handpos;
MoveL t103, v100\V:=100.000, z1, wi_tGripper, \WObj:=handpos;
MoveL t104, v100\V:=100.000, z1, wi_tGripper, \WObj:=handpos;
MoveL t105, v100\V:=100.000, z1, wi_tGripper, \WObj:=handpos;
MoveL t106, v100\V:=100.000, z1, wi_tGripper, \WObj:=handpos;
MoveL t107, v100\V:=100.000, z1, wi_tGripper, \WObj:=handpos;
MoveL t108, v100\V:=100.000, z1, wi_tGripper, \WObj:=handpos;
MoveL t109, v100\V:=100.000, z1, wi_tGripper, \WObj:=handpos;
MoveL t110, v100\V:=100.000, z1, wi_tGripper, \WObj:=handpos;
MoveL t111, v100\V:=100.000, z1, wi_tGripper, \WObj:=handpos;
MoveL t112, v100\V:=100.000, z1, wi_tGripper, \WObj:=handpos;
MoveL t113, v100\V:=100.000, z1, wi_tGripper, \WObj:=handpos;
MoveL t114, v100\V:=100.000, z1, wi_tGripper, \WObj:=handpos;
MoveL t115, v100\V:=100.000, z1, wi_tGripper, \WObj:=handpos;
MoveL t116, v100\V:=100.000, z1, wi_tGripper, \WObj:=handpos;
MoveL t117, v100\V:=100.000, z1, wi_tGripper, \WObj:=handpos;
MoveL t118, v100\V:=100.000, z1, wi_tGripper, \WObj:=handpos;
MoveL t119, v100\V:=100.000, z1, wi_tGripper, \WObj:=handpos;
MoveL t120, v100\V:=100.000, z1, wi_tGripper, \WObj:=handpos;
MoveL t121, v100\V:=100.000, z1, wi_tGripper, \WObj:=handpos;
MoveL t122, v100\V:=100.000, z1, wi_tGripper, \WObj:=handpos;
MoveL t123, v100\V:=100.000, z1, wi_tGripper, \WObj:=handpos;
MoveL t124, v100\V:=100.000, z1, wi_tGripper, \WObj:=handpos;
MoveL t125, v100\V:=100.000, z1, wi_tGripper, \WObj:=handpos;
MoveL t126, v100\V:=100.000, z1, wi_tGripper, \WObj:=handpos;
MoveL t127, v100\V:=100.000, z1, wi_tGripper, \WObj:=handpos;
MoveL t128, v100\V:=100.000, z1, wi_tGripper, \WObj:=handpos;
MoveL t129, v100\V:=100.000, z1, wi_tGripper, \WObj:=handpos;
MoveL t130, v100\V:=100.000, z1, wi_tGripper, \WObj:=handpos;
MoveL t131, v100\V:=100.000, z1, wi_tGripper, \WObj:=handpos;
MoveL t132, v100\V:=100.000, z1, wi_tGripper, \WObj:=handpos;
MoveL t133, v100\V:=100.000, z1, wi_tGripper, \WObj:=handpos;
MoveL t134, v100\V:=100.000, z1, wi_tGripper, \WObj:=handpos;
MoveL t135, v100\V:=100.000, z1, wi_tGripper, \WObj:=handpos;
MoveL t136, v100\V:=100.000, z1, wi_tGripper, \WObj:=handpos;
MoveL t137, v100\V:=100.000, z1, wi_tGripper, \WObj:=handpos;
MoveL t138, v100\V:=100.000, z1, wi_tGripper, \WObj:=handpos;
MoveL t139, v100\V:=100.000, z1, wi_tGripper, \WObj:=handpos;
MoveL t140, v100\V:=100.000, z1, wi_tGripper, \WObj:=handpos;
MoveL t141, v100\V:=100.000, z1, wi_tGripper, \WObj:=handpos;
MoveL t142, v100\V:=100.000, z1, wi_tGripper, \WObj:=handpos;
MoveL t143, v100\V:=100.000, z1, wi_tGripper, \WObj:=handpos;
MoveL t144, v100\V:=100.000, z1, wi_tGripper, \WObj:=handpos;
MoveL t145, v100\V:=100.000, z1, wi_tGripper, \WObj:=handpos;
MoveL t146, v100\V:=100.000, z1, wi_tGripper, \WObj:=handpos;
MoveL t147, v100\V:=100.000, z1, wi_tGripper, \WObj:=handpos;
MoveL t148, v100\V:=100.000, z1, wi_tGripper, \WObj:=handpos;
MoveL t149, v100\V:=100.000, z1, wi_tGripper, \WObj:=handpos;
MoveL t150, v100\V:=100.000, z1, wi_tGripper, \WObj:=handpos;
MoveL t151, v100\V:=100.000, z1, wi_tGripper, \WObj:=handpos;
MoveL t152, v100\V:=100.000, z1, wi_tGripper, \WObj:=handpos;
MoveL t153, v100\V:=100.000, z1, wi_tGripper, \WObj:=handpos;
MoveL t154, v100\V:=100.000, z1, wi_tGripper, \WObj:=handpos;
MoveL t155, v100\V:=100.000, z1, wi_tGripper, \WObj:=handpos;
MoveL t156, v100\V:=100.000, z1, wi_tGripper, \WObj:=handpos;
MoveL t157, v100\V:=100.000, z1, wi_tGripper, \WObj:=handpos;
MoveL t158, v100\V:=100.000, z1, wi_tGripper, \WObj:=handpos;
MoveL t159, v100\V:=100.000, z1, wi_tGripper, \WObj:=handpos;
MoveL t160, v100\V:=100.000, z1, wi_tGripper, \WObj:=handpos;
MoveL t161, v100\V:=100.000, z1, wi_tGripper, \WObj:=handpos;
MoveL t162, v100\V:=100.000, z1, wi_tGripper, \WObj:=handpos;
MoveL t163, v100\V:=100.000, z1, wi_tGripper, \WObj:=handpos;
MoveL t164, v100\V:=100.000, z1, wi_tGripper, \WObj:=handpos;
MoveL t165, v100\V:=100.000, z1, wi_tGripper, \WObj:=handpos;
MoveL t166, v100\V:=100.000, z1, wi_tGripper, \WObj:=handpos;
MoveL t167, v100\V:=100.000, z1, wi_tGripper, \WObj:=handpos;
MoveL t168, v100\V:=100.000, z1, wi_tGripper, \WObj:=handpos;
MoveL t169, v100\V:=100.000, z1, wi_tGripper, \WObj:=handpos;
MoveL t170, v100\V:=100.000, z1, wi_tGripper, \WObj:=handpos;
MoveL t171, v100\V:=100.000, z1, wi_tGripper, \WObj:=handpos;
MoveL t172, v100\V:=100.000, z1, wi_tGripper, \WObj:=handpos;
MoveL t173, v100\V:=100.000, z1, wi_tGripper, \WObj:=handpos;
MoveL t174, v100\V:=100.000, z1, wi_tGripper, \WObj:=handpos;
MoveL t175, v100\V:=100.000, z1, wi_tGripper, \WObj:=handpos;
MoveL t176, v100\V:=100.000, z1, wi_tGripper, \WObj:=handpos;
MoveL t177, v100\V:=100.000, z1, wi_tGripper, \WObj:=handpos;
MoveL t178, v100\V:=100.000, z1, wi_tGripper, \WObj:=handpos;
MoveL t179, v100\V:=100.000, z1, wi_tGripper, \WObj:=handpos;
MoveL t180, v100\V:=100.000, z1, wi_tGripper, \WObj:=handpos;
MoveL t181, v100\V:=100.000, z1, wi_tGripper, \WObj:=handpos;
MoveL t182, v100\V:=100.000, z1, wi_tGripper, \WObj:=handpos;
MoveL t183, v100\V:=100.000, z1, wi_tGripper, \WObj:=handpos;
MoveL t184, v100\V:=100.000, z1, wi_tGripper, \WObj:=handpos;
MoveL t185, v100\V:=100.000, z1, wi_tGripper, \WObj:=handpos;
MoveL t186, v100\V:=100.000, z1, wi_tGripper, \WObj:=handpos;
MoveL t187, v100\V:=100.000, z1, wi_tGripper, \WObj:=handpos;
MoveL t188, v100\V:=100.000, z1, wi_tGripper, \WObj:=handpos;
MoveL t189, v100\V:=100.000, z1, wi_tGripper, \WObj:=handpos;
MoveL t190, v100\V:=100.000, z1, wi_tGripper, \WObj:=handpos;
MoveL t191, v100\V:=100.000, z1, wi_tGripper, \WObj:=handpos;
MoveL t192, v100\V:=100.000, z1, wi_tGripper, \WObj:=handpos;
MoveL t193, v100\V:=100.000, z1, wi_tGripper, \WObj:=handpos;
MoveL t194, v100\V:=100.000, z1, wi_tGripper, \WObj:=handpos;
MoveL t195, v100\V:=100.000, z1, wi_tGripper, \WObj:=handpos;
MoveL t196, v100\V:=100.000, z1, wi_tGripper, \WObj:=handpos;
MoveL t197, v100\V:=100.000, z1, wi_tGripper, \WObj:=handpos;
MoveL t198, v100\V:=100.000, z1, wi_tGripper, \WObj:=handpos;
MoveL t199, v100\V:=100.000, z1, wi_tGripper, \WObj:=handpos;

ENDPROC
ENDMODULE
